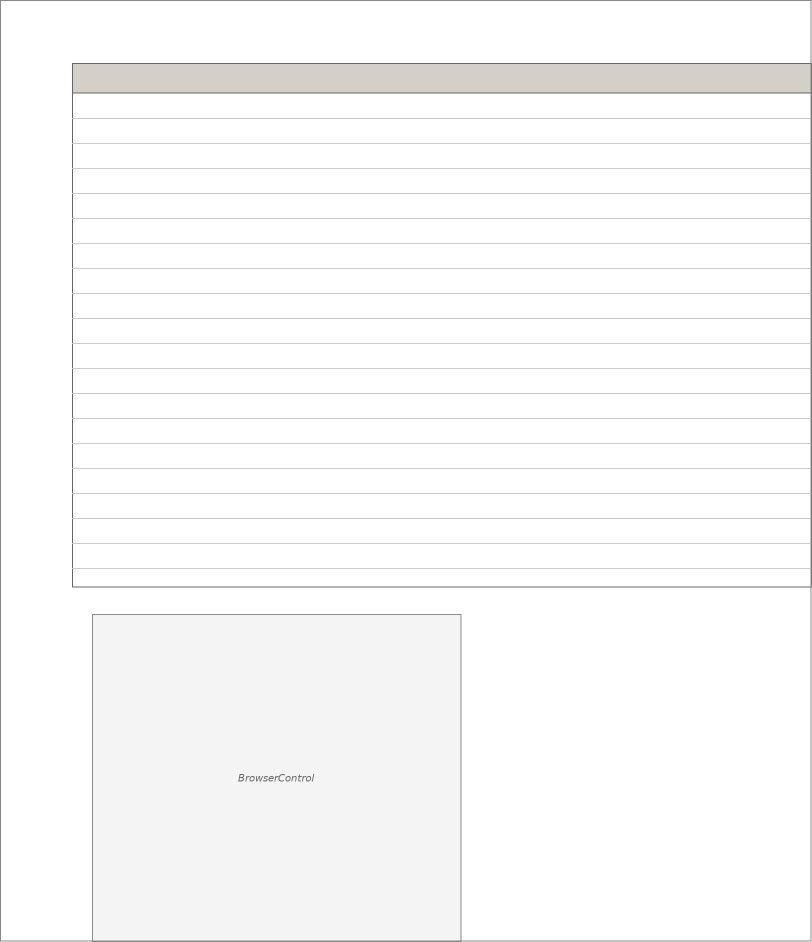
VISUALIZATION StateEthercat  // 812x942
    Table (72,63 740x524), data array: Tableau_Etat_Ethercat
        p3854506369: Tableau_Etat_Ethercat[INDEX].deviceState
        p1892666644: Tableau_Etat_Ethercat[INDEX].linkState
        p1014161805: 200 - 0 + INT#1
    BrowserControl (92,614 369x328)
        p3734058945: 'http://21.63.1.102/files/index.html#/dashboard/status'
        p2179181546: true
END_VISUALIZATION

(* stored: Version 1.1.0.1
   Visu StateEthercat: Id {88e33ae1-672d-4b77-86ea-7e6f0244af76} *)
